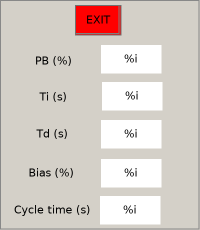
VISUALIZATION PidParameterMenu  // 200x230
    Textfield (100,44 62x30), "%i", text variable: PidParameterMenuBindings.PbTextField_TextVariable
        OnMouseDown: write the text variable via VisuDialogs.Numpad, min 1, max 999
    Label (2,39 103x44), "PB (%)"
    Button (75,5 46x30), "EXIT"
        toggle MainScreenBindings.PidParamMenuButton_ToggleVariable
    Label (2,75 103x44), "Ti (s)"
    Label (1,112 103x44), "Td (s)"
    Textfield (101,81 62x30), "%i", text variable: PidParameterMenuBindings.TiTextField_TextVariable
        OnMouseDown: write the text variable via VisuDialogs.Numpad, min 1, max 5999
    Textfield (100,119 62x30), "%i", text variable: PidParameterMenuBindings.TdTextField_TextVariable
        OnMouseDown: write the text variable via VisuDialogs.Numpad, min 1, max 5999
    Label (0,151 103x44), "Bias (%)"
    Textfield (100,158 62x30), "%i", text variable: PidParameterMenuBindings.BiasTextField_TextVariable
        OnMouseDown: write the text variable via VisuDialogs.Numpad, min 0, max 999
    Label (-6,188 117x44), "Cycle time (s)"
    Textfield (99,195 62x30), "%i", text variable: PidParameterMenuBindings.IterationTimeTextField_TextVariable
        OnMouseDown: write the text variable via VisuDialogs.Numpad, min 1, max 5999
END_VISUALIZATION

(* stored: Version 1.1.0.1, ProductVersion 3.1.4024.9
   Visu PidParameterMenu: Id {a703d9d6-e69e-4ef0-9cb6-83cbff51e043} *)
